// TIA Portal V15.1 export
// export: Created 2024-06-21T08:41:13.7762127Z, ExportSetting WithDefaults, DisplayName Totally Integrated Automation Portal, DisplayVersion V15.1 Update 5, DisplayName TIA Portal Openness, DisplayVersion V15.1 Update 5, DisplayName SINAMICS Startdrive Advanced, DisplayVersion V15.1, DisplayName G130, G150, S120, S150, SINAMICS MV, S210, DisplayVersion V15.1, DisplayName G110M, G120, G120C, G120D, G120P, DisplayVersion V15.1, DisplayName STEP 7 Professional, DisplayVersion V15.1 Update 5, DisplayName STEP 7 Safety, DisplayVersion V15.1, DisplayName WinCC Professional, DisplayVersion V15.1 Update 5, DisplayName SIMATIC Visualization Architect, DisplayVersion V15.1
FUNCTION_BLOCK "LGBGateMaint"   // FB6672, FBD
TITLE = LGBGateMaint
{ S7_Optimized_Access := 'TRUE' }
VERSION : 0.1
// ...
// stored: AutoNumber false, IsIECCheckEnabled false, IsRetainMemResEnabled false, MemoryReserve 100, SetENOAutomatically False, UDAEnableTagReadback false
   VAR_INPUT
      I_SafetyGateInput { ExternalAccessible := 'False'; ExternalVisible := 'False'; ExternalWritable := 'False'} : Bool;   // Input safety alarm (Summary door closed [T] and handle closed [R] - SK)
      I_Q { ExternalAccessible := 'False'; ExternalVisible := 'False'; ExternalWritable := 'False'} : Bool;   // Input Safety Logic Result Alarm (normally closed)
      I_EnableAlarm { ExternalAccessible := 'False'; ExternalVisible := 'False'; ExternalWritable := 'False'} : Bool := TRUE;   // Enable alarm from upper level
      I_LampTest { ExternalAccessible := 'False'; ExternalVisible := 'False'; ExternalWritable := 'False'} : Bool;   // Lamp test
      I_AutoMode { ExternalAccessible := 'False'; ExternalVisible := 'False'; ExternalWritable := 'False'} : Bool;   // Automatic mode active
      I_AccessStopReqPB { ExternalAccessible := 'False'; ExternalVisible := 'False'; ExternalWritable := 'False'} : Bool;   // Stop position reached for Request access / Access stop position reached
      I_AccessStopReached { ExternalAccessible := 'False'; ExternalVisible := 'False'; ExternalWritable := 'False'} : Bool;   // Stop position reached for Request access / Access stop position reached
      I_CycleStopPB { ExternalAccessible := 'False'; ExternalVisible := 'False'; ExternalWritable := 'False'} : Bool;   // CycleStop PB
      I_CycleStopReached { ExternalAccessible := 'False'; ExternalVisible := 'False'; ExternalWritable := 'False'} : Bool;   // Cycle stop reached
      I_MaintPassageReqPB { ExternalAccessible := 'False'; ExternalVisible := 'False'; ExternalWritable := 'False'} : Bool;   // Maintenance requestPB
      I_MaintPosReached { ExternalAccessible := 'False'; ExternalVisible := 'False'; ExternalWritable := 'False'} : Bool;   // Maintenance Position Reached
      I_AlarmABAct { ExternalAccessible := 'False'; ExternalVisible := 'False'; ExternalWritable := 'False'} : Bool;   // Alarm A or B active
   END_VAR
   VAR_OUTPUT
      O_MaintReq { ExternalAccessible := 'False'; ExternalVisible := 'False'; ExternalWritable := 'False'} : Bool;   // Switch Maintenance
      O_MaintPBInd { ExternalAccessible := 'False'; ExternalVisible := 'False'; ExternalWritable := 'False'} : Bool;   // MaintPB lamp
      O_CycleStopReq { ExternalAccessible := 'False'; ExternalVisible := 'False'; ExternalWritable := 'False'} : Bool;   // Request for cycle stop / Request for Cycle Stop
      O_CycleStopPBInd { ExternalAccessible := 'False'; ExternalVisible := 'False'; ExternalWritable := 'False'} : Bool;   // CycleStopPB lamp
      O_AccesStopReq { ExternalAccessible := 'False'; ExternalVisible := 'False'; ExternalWritable := 'False'} : Bool;   // Request for cycle stop / Request for Cycle Stop / Request for Acces Stop Indication / Request for Access
      O_AccesStopReqPBInd { ExternalAccessible := 'False'; ExternalVisible := 'False'; ExternalWritable := 'False'} : Bool;   // Request for Acces Stop
      O_AccessReqAlarm { ExternalAccessible := 'False'; ExternalVisible := 'False'; ExternalWritable := 'False'} : Bool;   // Request for Acces Stop Alarm
   END_VAR
   VAR_IN_OUT
      IO_Alarm : "Alarm";   // Alarm
      H_HMI : "H_HMI";   // Animation
      "H_GateLock-MGB" : "H_GateMaint";   // Animation
   END_VAR
   VAR
      DelayStop { ExternalAccessible := 'False'; ExternalVisible := 'False'; ExternalWritable := 'False'} : Bool;   // Stop pushbutton delayed
      DelayMaint { ExternalAccessible := 'False'; ExternalVisible := 'False'; ExternalWritable := 'False'} : Bool;   // Maintenance pushbutton delayed
      SafetyGateAlarm { ExternalAccessible := 'False'; ExternalVisible := 'False'; ExternalWritable := 'False'} : Bool;   // Alarm / Safety Gate Alarm
      AccessReqAlarm { ExternalAccessible := 'False'; ExternalVisible := 'False'; ExternalWritable := 'False'} : Bool;   // Alarm / Solenoid Alarm / Access Request Alarm
      AccessReqSel { ExternalAccessible := 'False'; ExternalVisible := 'False'; ExternalWritable := 'False'} : Bool;   // Request access memory / Request access selected
      AccessReq { ExternalAccessible := 'False'; ExternalVisible := 'False'; ExternalWritable := 'False'} : Bool;   // Request access memory / Request access
      AccessReqMaintSel { ExternalAccessible := 'False'; ExternalVisible := 'False'; ExternalWritable := 'False'} : Bool;   // Request access maint memory
      MaintReq { ExternalAccessible := 'False'; ExternalVisible := 'False'; ExternalWritable := 'False'} : Bool;   // Request access maint memory
      CycleReq { ExternalAccessible := 'False'; ExternalVisible := 'False'; ExternalWritable := 'False'} : Bool;   // Request access cycle memory
      AccessReqCycleSel { ExternalAccessible := 'False'; ExternalVisible := 'False'; ExternalWritable := 'False'} : Bool;   // Request access cycle memory
      NotAutoMem { ExternalAccessible := 'False'; ExternalVisible := 'False'; ExternalWritable := 'False'} : Bool;   // Pushbutton stop memory
      DelayTimerPbStop { ExternalAccessible := 'False'; ExternalVisible := 'False'; ExternalWritable := 'False'} : IEC_TIMER;   // Delay timer for Stop pushbutton
      DelayTimerMaintPb { ExternalAccessible := 'False'; ExternalVisible := 'False'; ExternalWritable := 'False'} : IEC_TIMER;   // Delay timer for maintenance pushbutton
      Edge { ExternalAccessible := 'False'; ExternalVisible := 'False'; ExternalWritable := 'False'} : Array[1..15] of Bool;   // Edges / Edge
      _ToggleReqAccess { ExternalAccessible := 'False'; ExternalVisible := 'False'; ExternalWritable := 'False'} : "LToggle";   // Toggle request access / Toggle access request
      _ToggleReqAccessMaint { ExternalAccessible := 'False'; ExternalVisible := 'False'; ExternalWritable := 'False'} : "LToggle";   // Toggle request access
      _ToggleReqAccessCycle { ExternalAccessible := 'False'; ExternalVisible := 'False'; ExternalWritable := 'False'} : "LToggle";   // Toggle request access
      IEC_Timer_0_Instance { ExternalAccessible := 'False'; ExternalVisible := 'False'; ExternalWritable := 'False'} : IEC_TIMER;
   END_VAR
   VAR_TEMP   // added for the SCL form of the ladder/FBD networks
      _w1 : Bool;
      _w2 : Bool;
      _w3 : Bool;
      _w4 : Bool;
   END_VAR
BEGIN

REGION Network 1: **** 2.2 - Alarms - Alarms Generation **** Solenoid Alarm / **** 2.2 - Alarms - Alarms Generation **** Safety Gate Alarm
   // Solenoid alarm / Condition of the Safety Alarm for the Normal Closed input
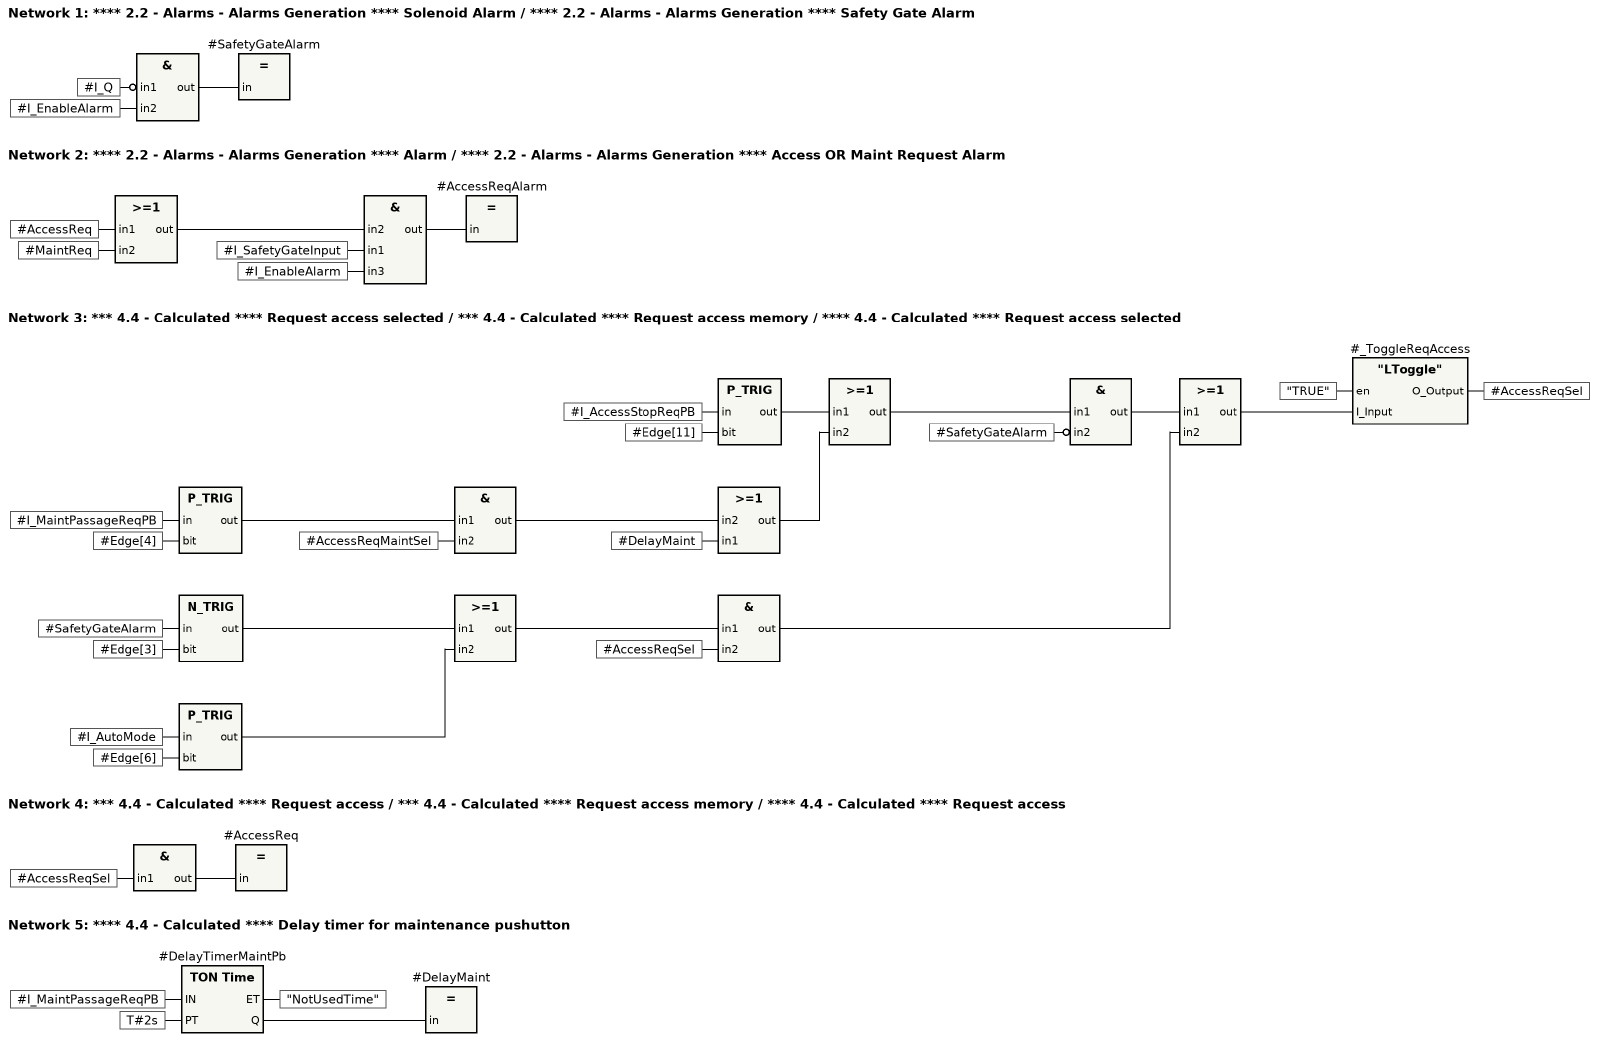
   #SafetyGateAlarm := NOT #I_Q AND #I_EnableAlarm;
END_REGION

REGION Network 2: **** 2.2 - Alarms - Alarms Generation **** Alarm / **** 2.2 - Alarms - Alarms Generation **** Access OR Maint Request Alarm
   // Creation of the Safety Alarm for the Normal Closed input / Alarm to notify that an access to the line is requested at the gate
   #AccessReqAlarm := (#AccessReq OR #MaintReq) AND #I_SafetyGateInput AND #I_EnableAlarm;
END_REGION

REGION Network 3: *** 4.4 - Calculated **** Request access selected / *** 4.4 - Calculated **** Request access memory / **** 4.4 - Calculated **** Request access selected
   // Request access selected / Request access memory
   #_w1 := #I_AccessStopReqPB AND NOT #Edge[11];   // rising edge
   #Edge[11] := #I_AccessStopReqPB;
   #_w2 := #I_MaintPassageReqPB AND NOT #Edge[4];   // rising edge
   #Edge[4] := #I_MaintPassageReqPB;
   #_w3 := NOT #SafetyGateAlarm AND #Edge[3];   // falling edge
   #Edge[3] := #SafetyGateAlarm;
   #_w4 := #I_AutoMode AND NOT #Edge[6];   // rising edge
   #Edge[6] := #I_AutoMode;
   IF "TRUE" THEN
       #_ToggleReqAccess(I_Input := ((#_w1 OR (#_w2 AND #AccessReqMaintSel) OR #DelayMaint) AND NOT #SafetyGateAlarm) OR ((#_w3 OR #_w4) AND #AccessReqSel),   // "LToggle"
                         O_Output => #AccessReqSel);
   END_IF;
END_REGION

REGION Network 4: *** 4.4 - Calculated **** Request access / *** 4.4 - Calculated **** Request access memory / **** 4.4 - Calculated **** Request access
   // Request access / Request access memory
   #AccessReq := #AccessReqSel;
END_REGION

REGION Network 5: **** 4.4 - Calculated **** Delay timer for maintenance pushutton
   // Delay timer for maintenance pushutton
   #DelayTimerMaintPb.TON(IN := #I_MaintPassageReqPB, PT := T#2s, ET => "NotUsedTime");
   #DelayMaint := #DelayTimerMaintPb.Q;
END_REGION

REGION Network 6: *** 4.4 - Calculated **** Request access selected / *** 4.4 - Calculated **** Request access memory / **** 4.4 - Calculated **** Request maint access selected
   // Request access selected / Request access memory
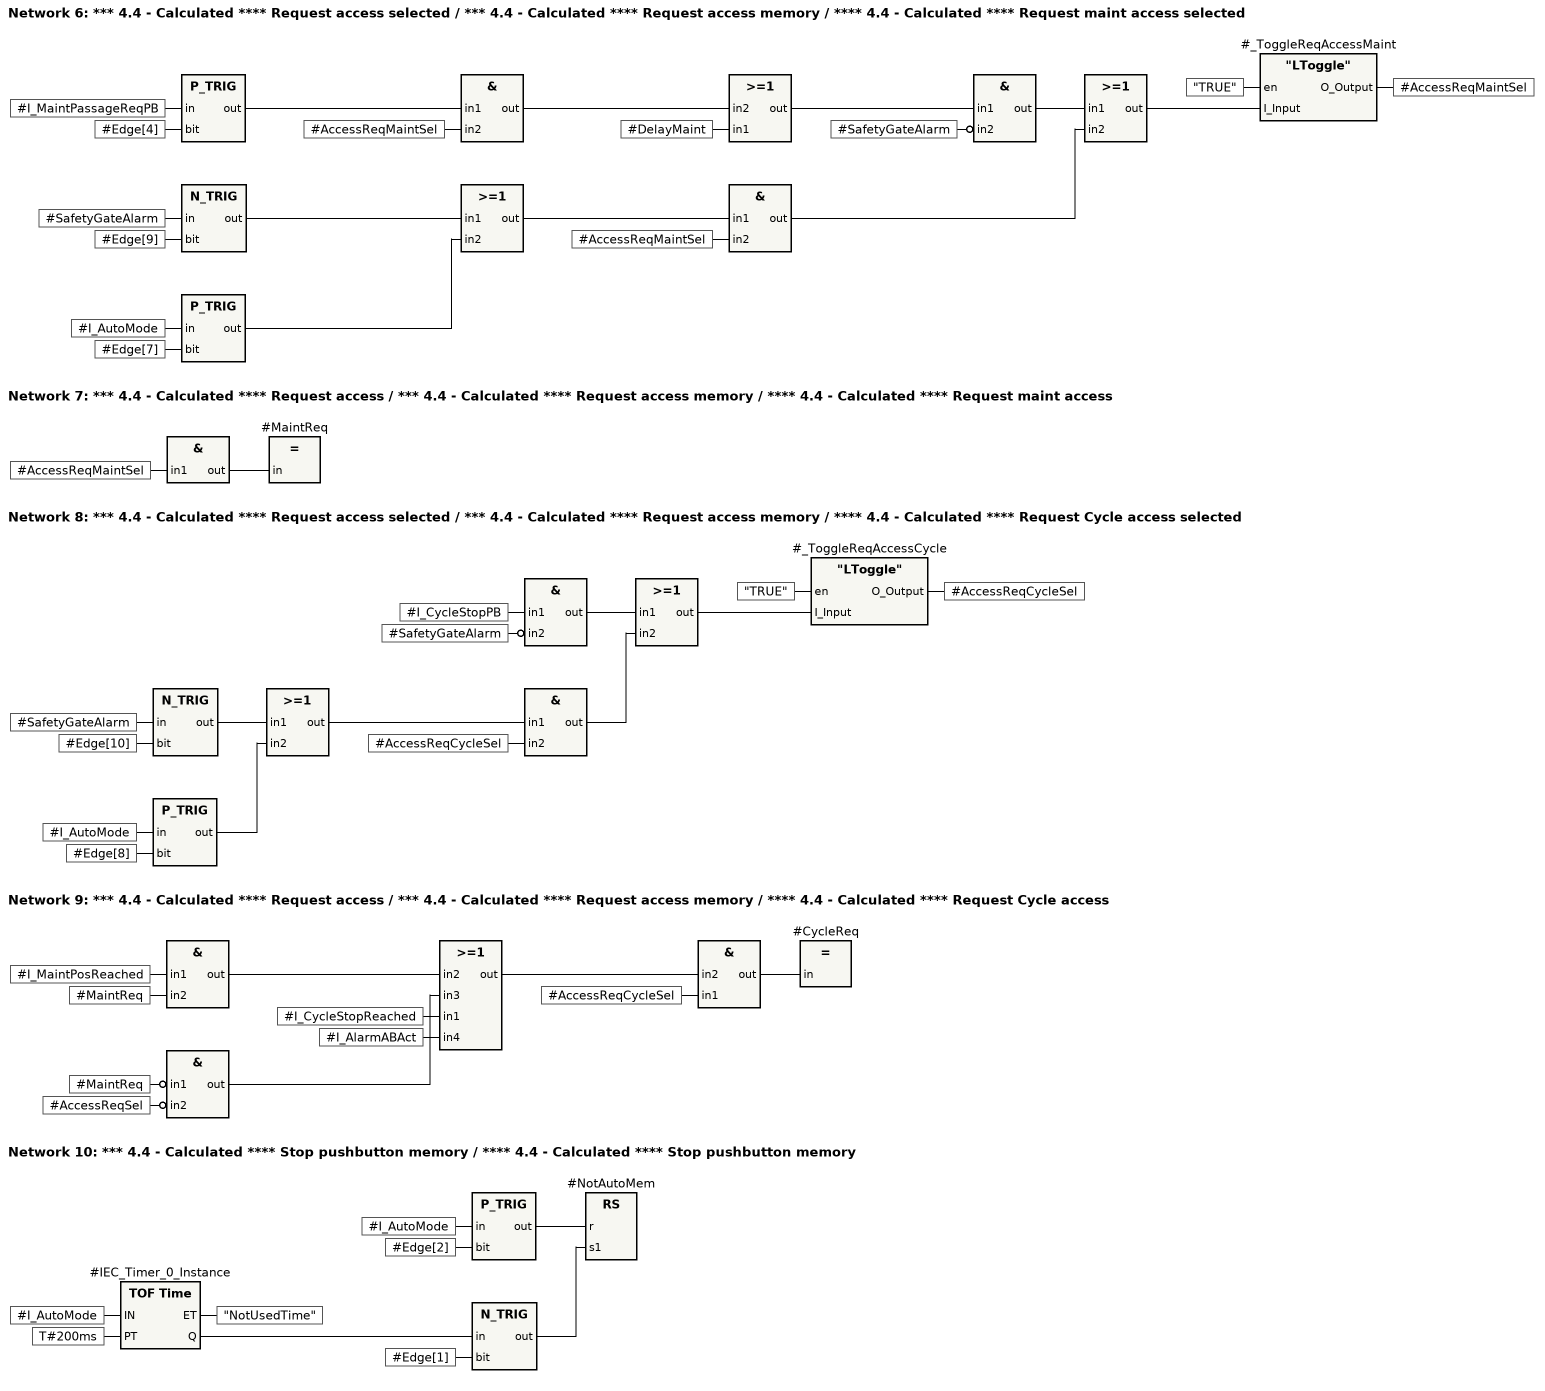
   #_w1 := #I_MaintPassageReqPB AND NOT #Edge[4];   // rising edge
   #Edge[4] := #I_MaintPassageReqPB;
   #_w2 := NOT #SafetyGateAlarm AND #Edge[9];   // falling edge
   #Edge[9] := #SafetyGateAlarm;
   #_w3 := #I_AutoMode AND NOT #Edge[7];   // rising edge
   #Edge[7] := #I_AutoMode;
   IF "TRUE" THEN
       #_ToggleReqAccessMaint(I_Input := (((#_w1 AND #AccessReqMaintSel) OR #DelayMaint) AND NOT #SafetyGateAlarm) OR ((#_w2 OR #_w3) AND #AccessReqMaintSel),   // "LToggle"
                              O_Output => #AccessReqMaintSel);
   END_IF;
END_REGION

REGION Network 7: *** 4.4 - Calculated **** Request access / *** 4.4 - Calculated **** Request access memory / **** 4.4 - Calculated **** Request maint access
   // Request access / Request access memory / Request maint access
   #MaintReq := #AccessReqMaintSel;
END_REGION

REGION Network 8: *** 4.4 - Calculated **** Request access selected / *** 4.4 - Calculated **** Request access memory / **** 4.4 - Calculated **** Request Cycle access selected
   // Request access selected / Request access memory / Request cycle access selected
   #_w1 := NOT #SafetyGateAlarm AND #Edge[10];   // falling edge
   #Edge[10] := #SafetyGateAlarm;
   #_w2 := #I_AutoMode AND NOT #Edge[8];   // rising edge
   #Edge[8] := #I_AutoMode;
   IF "TRUE" THEN
       #_ToggleReqAccessCycle(I_Input := (#I_CycleStopPB AND NOT #SafetyGateAlarm) OR ((#_w1 OR #_w2) AND #AccessReqCycleSel),   // "LToggle"
                              O_Output => #AccessReqCycleSel);
   END_IF;
END_REGION

REGION Network 9: *** 4.4 - Calculated **** Request access / *** 4.4 - Calculated **** Request access memory / **** 4.4 - Calculated **** Request Cycle access
   // Request access / Request access memory / Request cycle access
   #CycleReq := ((#I_MaintPosReached AND #MaintReq) OR (NOT #MaintReq AND NOT #AccessReqSel) OR #I_CycleStopReached OR #I_AlarmABAct) AND #AccessReqCycleSel;
END_REGION

REGION Network 10: *** 4.4 - Calculated **** Stop pushbutton memory / **** 4.4 - Calculated **** Stop pushbutton memory
   // Stop pushbutton memory
   #_w1 := #I_AutoMode AND NOT #Edge[2];   // rising edge
   #Edge[2] := #I_AutoMode;
   #IEC_Timer_0_Instance.TOF(IN := #I_AutoMode, PT := T#200ms, ET => "NotUsedTime");
   #_w2 := NOT #IEC_Timer_0_Instance.Q AND #Edge[1];   // falling edge
   #Edge[1] := #IEC_Timer_0_Instance.Q;
   IF #_w1 THEN
       #NotAutoMem := FALSE;   // RS flip-flop
   END_IF;
   IF #_w2 THEN #NotAutoMem := TRUE; END_IF;
END_REGION

REGION Network 11: *** 4.4 - Calculated **** Delay timer stop pushbutton / **** 4.4 - Calculated **** Delay timer stop pushbutton
   // Delay for Stop pushbutton
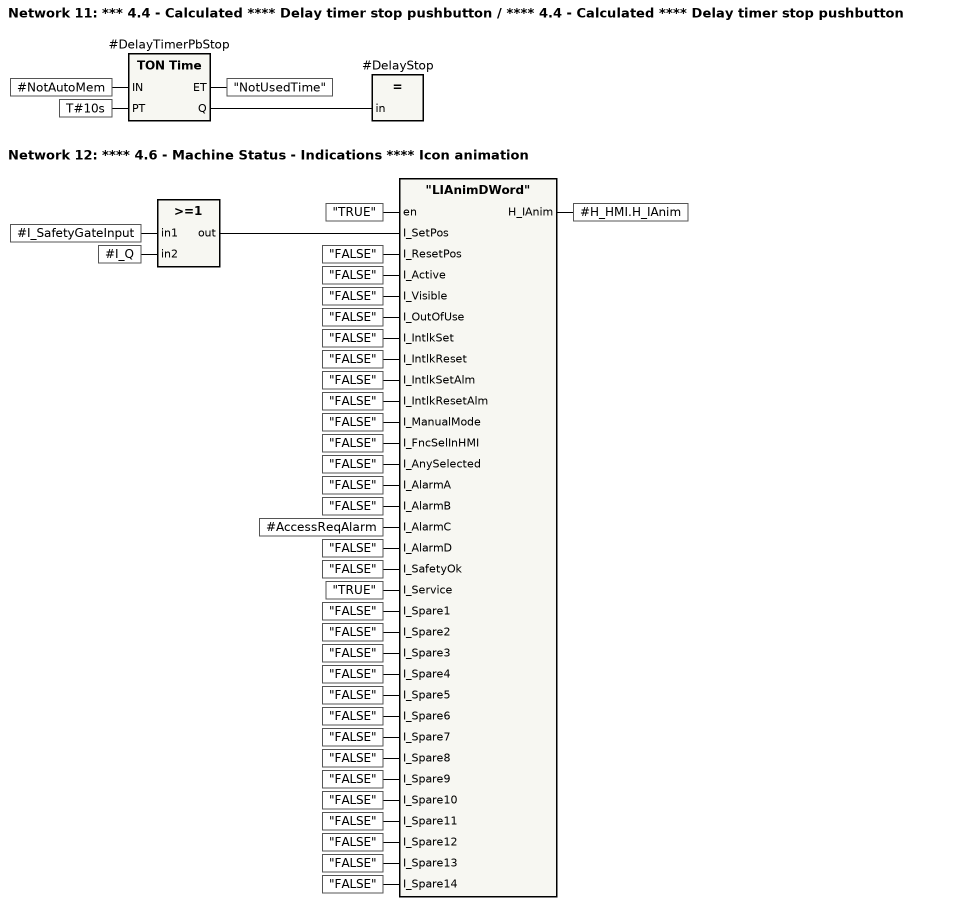
   #DelayTimerPbStop.TON(IN := #NotAutoMem, PT := T#10s, ET => "NotUsedTime");
   #DelayStop := #DelayTimerPbStop.Q;
END_REGION

REGION Network 12: **** 4.6 - Machine Status - Indications **** Icon animation
   // Icon Animation
   IF "TRUE" THEN
       "LIAnimDWord"(I_SetPos := #I_SafetyGateInput OR #I_Q,
                     I_ResetPos := "FALSE",
                     I_Active := "FALSE",
                     I_Visible := "FALSE",
                     I_OutOfUse := "FALSE",
                     I_IntlkSet := "FALSE",
                     I_IntlkReset := "FALSE",
                     I_IntlkSetAlm := "FALSE",
                     I_IntlkResetAlm := "FALSE",
                     I_ManualMode := "FALSE",
                     I_FncSelInHMI := "FALSE",
                     I_AnySelected := "FALSE",
                     I_AlarmA := "FALSE",
                     I_AlarmB := "FALSE",
                     I_AlarmC := #AccessReqAlarm,
                     I_AlarmD := "FALSE",
                     I_SafetyOk := "FALSE",
                     I_Service := "TRUE",
                     I_Spare1 := "FALSE",
                     I_Spare2 := "FALSE",
                     I_Spare3 := "FALSE",
                     I_Spare4 := "FALSE",
                     I_Spare5 := "FALSE",
                     I_Spare6 := "FALSE",
                     I_Spare7 := "FALSE",
                     I_Spare8 := "FALSE",
                     I_Spare9 := "FALSE",
                     I_Spare10 := "FALSE",
                     I_Spare11 := "FALSE",
                     I_Spare12 := "FALSE",
                     I_Spare13 := "FALSE",
                     I_Spare14 := "FALSE",
                     H_IAnim => #H_HMI.H_IAnim);
   END_IF;
END_REGION

REGION Network 13: **** 4.6 - Machine Status - Indications **** Animation
   // Animation
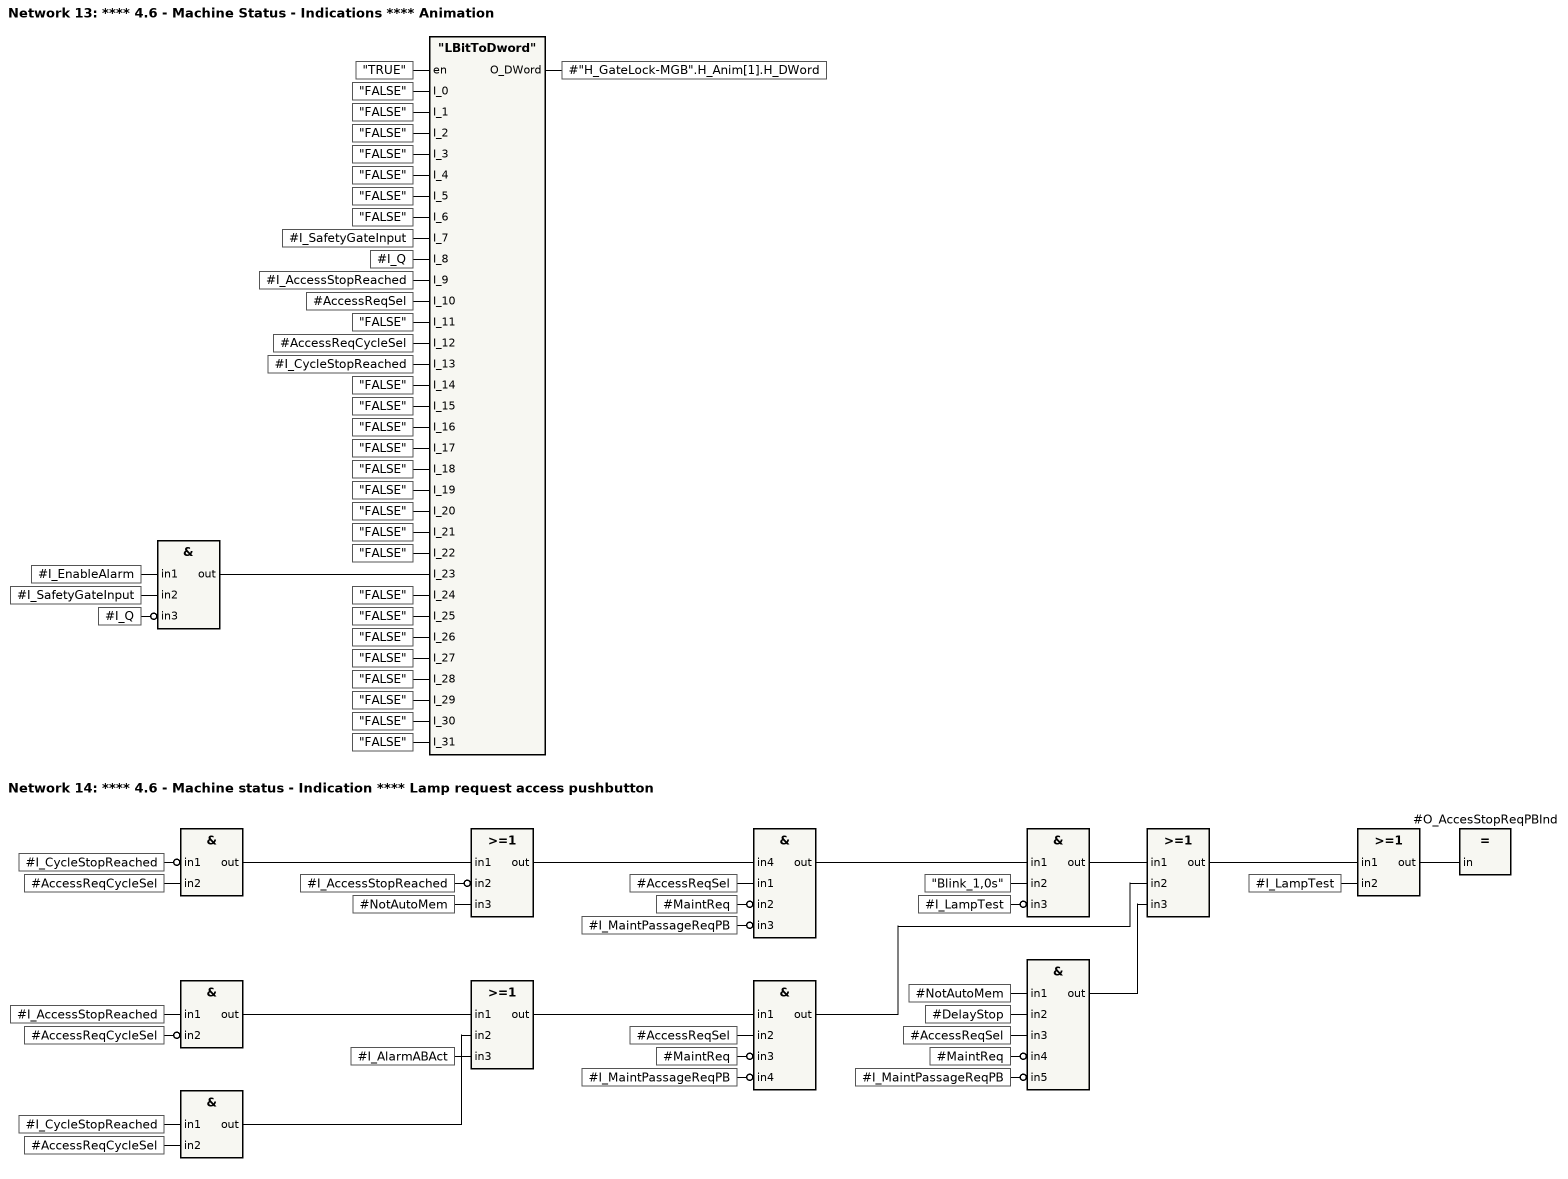
   IF "TRUE" THEN
       "LBitToDword"(I_0 := "FALSE",
                     I_1 := "FALSE",
                     I_2 := "FALSE",
                     I_3 := "FALSE",
                     I_4 := "FALSE",
                     I_5 := "FALSE",
                     I_6 := "FALSE",
                     I_7 := #I_SafetyGateInput,
                     I_8 := #I_Q,
                     I_9 := #I_AccessStopReached,
                     I_10 := #AccessReqSel,
                     I_11 := "FALSE",
                     I_12 := #AccessReqCycleSel,
                     I_13 := #I_CycleStopReached,
                     I_14 := "FALSE",
                     I_15 := "FALSE",
                     I_16 := "FALSE",
                     I_17 := "FALSE",
                     I_18 := "FALSE",
                     I_19 := "FALSE",
                     I_20 := "FALSE",
                     I_21 := "FALSE",
                     I_22 := "FALSE",
                     I_23 := #I_EnableAlarm AND #I_SafetyGateInput AND NOT #I_Q,
                     I_24 := "FALSE",
                     I_25 := "FALSE",
                     I_26 := "FALSE",
                     I_27 := "FALSE",
                     I_28 := "FALSE",
                     I_29 := "FALSE",
                     I_30 := "FALSE",
                     I_31 := "FALSE",
                     O_DWord => #"H_GateLock-MGB".H_Anim[1].H_DWord);
   END_IF;
END_REGION

REGION Network 14: **** 4.6 - Machine status - Indication **** Lamp request access pushbutton
   // Request Acces PB indication
   #O_AccesStopReqPBInd := (((NOT #I_CycleStopReached AND #AccessReqCycleSel) OR NOT #I_AccessStopReached OR #NotAutoMem) AND #AccessReqSel AND NOT #MaintReq AND NOT #I_MaintPassageReqPB AND "Blink_1,0s" AND NOT #I_LampTest) OR (((#I_AccessStopReached AND NOT #AccessReqCycleSel) OR (#I_CycleStopReached AND #AccessReqCycleSel) OR #I_AlarmABAct) AND #AccessReqSel AND NOT #MaintReq AND NOT #I_MaintPassageReqPB) OR (#NotAutoMem AND #DelayStop AND #AccessReqSel AND NOT #MaintReq AND NOT #I_MaintPassageReqPB) OR #I_LampTest;
END_REGION

REGION Network 15: **** 4.6 - Machine status - Indication **** Lamp Maintenance / reset safety / **** 4.6 - Machine status - Indication **** Lamp Maintenance/End switch / **** 4.6 - Machine status - Indication **** Lamp Maintenance
   // Maintenance/End SW indication / Maintenance Pb indication
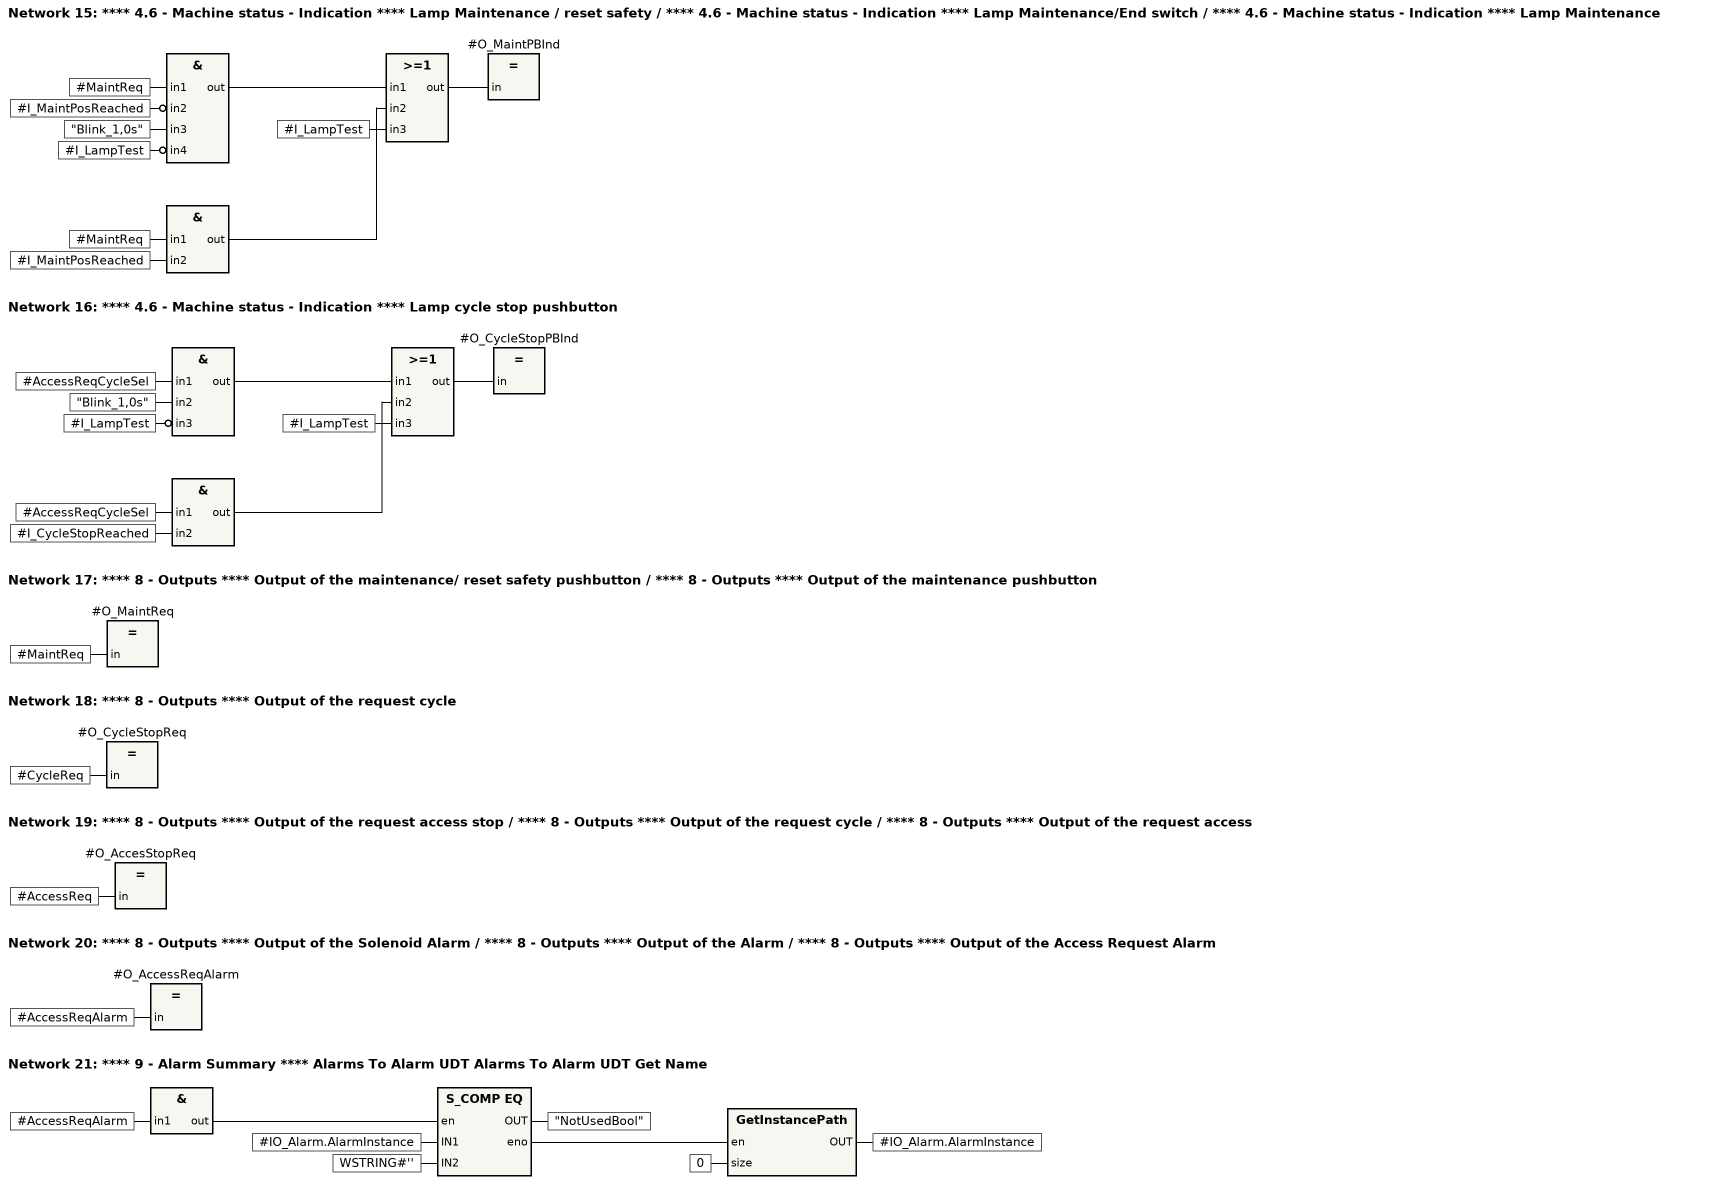
   #O_MaintPBInd := (#MaintReq AND NOT #I_MaintPosReached AND "Blink_1,0s" AND NOT #I_LampTest) OR (#MaintReq AND #I_MaintPosReached) OR #I_LampTest;
END_REGION

REGION Network 16: **** 4.6 - Machine status - Indication **** Lamp cycle stop pushbutton
   // Cycle Stop PB indication
   #O_CycleStopPBInd := (#AccessReqCycleSel AND "Blink_1,0s" AND NOT #I_LampTest) OR (#AccessReqCycleSel AND #I_CycleStopReached) OR #I_LampTest;
END_REGION

REGION Network 17: **** 8 - Outputs **** Output of the maintenance/ reset safety pushbutton / **** 8 - Outputs **** Output of the maintenance pushbutton
   // Output of the maintenance/ reset safety pushbutton / Output of the maintenance pushbutton
   #O_MaintReq := #MaintReq;
END_REGION

REGION Network 18: **** 8 - Outputs **** Output of the request cycle
   // Output of the request cycle
   #O_CycleStopReq := #CycleReq;
END_REGION

REGION Network 19: **** 8 - Outputs **** Output of the request access stop / **** 8 - Outputs **** Output of the request cycle / **** 8 - Outputs **** Output of the request access
   // Output of the request access stop / Output of the request cycle / Output of the request access
   #O_AccesStopReq := #AccessReq;
END_REGION

REGION Network 20: **** 8 - Outputs **** Output of the Solenoid Alarm / **** 8 - Outputs **** Output of the Alarm / **** 8 - Outputs **** Output of the Access Request Alarm
   // Output of the Solenoid Alarm / Output of the Alarm / Output of the Access Request Alarm
   #O_AccessReqAlarm := #AccessReqAlarm;
END_REGION

REGION Network 21: **** 9 - Alarm Summary **** Alarms To Alarm UDT Alarms To Alarm UDT Get Name
   // Alarm / Alarm D
   S_COMP(EN := #AccessReqAlarm,
          IN1 := #IO_Alarm.AlarmInstance,
          IN2 := WSTRING#'',
          OUT => "NotUsedBool",
          ENO => #_w1);
   IF #_w1 THEN GetInstancePath(size := 0, OUT => #IO_Alarm.AlarmInstance); END_IF;
END_REGION

REGION Network 22: **** 9 - Alarm Summary **** Alarms To Alarm UDT
   // Alarm / Alarm D
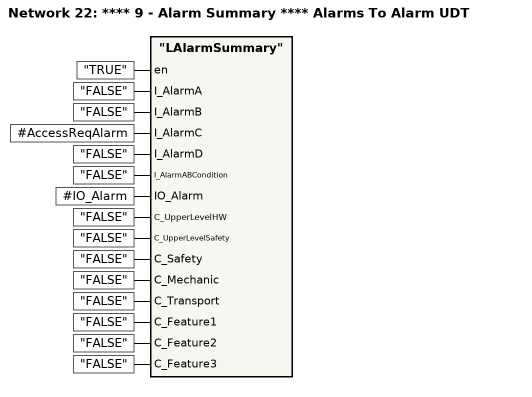
   IF "TRUE" THEN
       "LAlarmSummary"(I_AlarmA := "FALSE",
                       I_AlarmB := "FALSE",
                       I_AlarmC := #AccessReqAlarm,
                       I_AlarmD := "FALSE",
                       I_AlarmABCondition := "FALSE",
                       IO_Alarm := #IO_Alarm,
                       C_UpperLevelHW := "FALSE",
                       C_UpperLevelSafety := "FALSE",
                       C_Safety := "FALSE",
                       C_Mechanic := "FALSE",
                       C_Transport := "FALSE",
                       C_Feature1 := "FALSE",
                       C_Feature2 := "FALSE",
                       C_Feature3 := "FALSE");
   END_IF;
END_REGION
END_FUNCTION_BLOCK
